# B&R Automation Studio project Prak3
Automation Studio 4.5.2.102

## Configuration Config1

### Task classes (Cpu.sw)
```
Cyclic#4:
  Program <- Program.prg
VcDataObjects: Visu <- Visu.dob
Libraries: McBase, Library
```

### Hardware
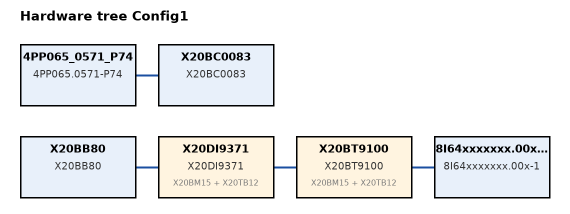
```
4PP065_0571_P74 : 4PP065.0571-P74 v1.1.2.0
  Connector IF5:
    ActivateDevice = 1
    Mode = Manual
    InternetAddress = 10.0.1.10
    SubnetMask = 255.255.255.0
  ConfigurationID = labBR
  VcObjectName = Visu
8I64xxxxxxx.00x-1 : 8I64xxxxxxx.00x-1 v2.1.3.0  [X2X1 -> X20BT9100.X2X1 [Cable Type=X2XCable, Length=10, Version=1.0.0.2]]
  FunctionModel = Standard
  packedETAD = packed
  packedCMDD = packed
X20BB80 : X20BB80 v1.0.2.0
X20BC0083 : X20BC0083 v2.14.0.0  [PLK1 -> 4PP065_0571_P74.IF4 (NodeNumber=2) [Cable Type=PowerlinkCable, Length=10, Version=1.0.0.2]; SL -> X20BB80.SL1]
X20BM15 : X20BM15 v1.0.1.0  [X2X1 -> X20BB80.IF1 (NodeNumber=5)]
X20BM15a : X20BM15 v1.0.1.0  [X2X1 -> X20BM15.X2X2 (NodeNumber=10)]
X20BT9100 : X20BT9100 v1.0.3.0  [SS1 -> X20TB12a.SS; SL -> X20BM15a.SL1]
X20DI9371 : X20DI9371 v1.0.2.0  [SS1 -> X20TB12.SS; SL -> X20BM15.SL1]
X20TB12 : X20TB12 v1.0.0.0
X20TB12a : X20TB12 v1.0.0.0
```

### IoMap.iom - 4PP065_0571_P74/IoMap.iom
```iecst
VAR_CONFIG
	::CMDD AT %QW."8I64xxxxxxx.00x-1".CMDD_Output;
	::ETAD AT %IW."8I64xxxxxxx.00x-1".ETAD_Input;
	::OTR AT %IW."8I64xxxxxxx.00x-1".OTR_Input;
	::LCR AT %IW."8I64xxxxxxx.00x-1".LCR_Input;
	::Speed AT %QW."8I64xxxxxxx.00x-1".LFRD_Output;
	::RUN AT %IX."X20DI9371".DigitalInput01;
END_VAR
```

## Logical view

### Global.var
```iecst
VAR
	ETAD : UINT;
	CMDD : UINT;
	Speed : INT;
	LCR : UINT;
	OTR : INT;
	RUN : BOOL;
END_VAR
```

### Program Logical/Program

#### Variables.var
```iecst
VAR
	STATE : UINT;
	speedDown : BOOL;
	speedUp : BOOL;
	Reset : BOOL;
	Onlinerun : USINT;
END_VAR
```

#### Main.c
```c
#include <bur/plctypes.h>

#ifdef _DEFAULT_INCLUDES
	#include <AsDefault.h>
#endif

void _INIT ProgramInit(void)
{
Speed=500;
}
BOOL up=0;
BOOL down=0;
void _CYCLIC ProgramCyclic(void)
{
	STATE=ETAD & 0x6f;
	if(RUN || Onlinerun){
		switch(STATE){
			case 64:
				CMDD=6;
				break;
			case 33:
				CMDD=15;
				break;
		}
	}
	else{
		CMDD=6;
	}
	if(speedUp==1 && up==0){
		Speed+=50;
		up=1;
	}
	if(speedUp==0){up=0;}

	if(speedDown==1 && down==0){
		Speed-=50;
		down=1;
	}
	if(speedDown==0){down=0;}
	if(OTR>8){
		while(Reset==0){
			RUN=0;
			Onlinerun=0;
		}
	}}

void _EXIT ProgramExit(void)
{

}
```
